TYPE ST_SiftError :
STRUCT
	bError : BOOL;     // True is this is an error. 
	nErrId : UDINT;    // The ID of this error.
	sReason : STRING;  // Error message in string format.
END_STRUCT
END_TYPE

(* stored: Version 1.1.0.1
   DUT ST_SiftError: Id {a683186e-ad47-4198-a1bb-0226db3e164a} *)
